// TIA Portal V17 export
// export: Created 2023-12-22T15:04:45.0691271Z, ExportSetting WithDefaults, DisplayName Totally Integrated Automation Portal, DisplayVersion V17, DisplayName TIA Portal Openness, DisplayVersion V17, DisplayName TIA Portal Version Control Interface, DisplayVersion V17, DisplayName STEP 7 Professional, DisplayVersion V17, DisplayName STEP 7 Safety, DisplayVersion V17, DisplayName WinCC Advanced, DisplayVersion V17
DATA_BLOCK "Main_Logick_DB"   // DB1
VERSION : 0.1
// stored: AutoNumber true, DBAccessibleFromOPCUA true, InstanceOfName Main_Logick, InstanceOfType FB
"Main_Logick"
   // VAR RETAIN
   //    Start : Bool;
   //    Start_Local : Bool;
   //    REQ_Pump : Bool;
   //    ev : Bool;
   //    Ready : Bool;
   //    Local : Bool;
   //    Mode : Bool;
   //    SP_Pump { S7_SetPoint := 'True'} : Real := 0.0;
   //    RM : Real;
   //    RM_SP { S7_SetPoint := 'True'} : Real := 0.0;
   //    Level_Norm { S7_SetPoint := 'True'} : Real := 50.0;
   //    Distance { S7_SetPoint := 'True'} : Real := 500.0;
   //    LE_Bar : Real;
   //    LE_Skvaz { S7_SetPoint := 'True'} : Real := 100.0;
   //    LE_Skvaz_RCHV { S7_SetPoint := 'True'} : Real := 0.0;
   //    Effect : Real;
   //    Alarm : Word;
   //    Alarms : Struct
   //       Leak : Bool;
   //       Level_Norm : Bool;
   //       LE_Warning : Bool;
   //       LE_Alarm : Bool;
   //    END_STRUCT;
   //    PID_Pump { S7_SetPoint := 'True'} : "PID_ex";
   // END_VAR
BEGIN
   PID_Pump.CMD.Vector := FALSE;
   PID_Pump.x := 1.0;
   PID_Pump.Settings.SP_P := 1.5;
   PID_Pump.Settings.SP_Ti := 150.0;
   PID_Pump.Settings.SP_Td := 0.0;
   PID_Pump.Settings.SP_Cycle := 0.2;
   PID_Pump.Settings.Max_SP := 500.0;
   PID_Pump.Settings.Min_SP := -500.0;
   PID_Pump.Settings.Max_in := 500.0;
   PID_Pump.Settings.Min_in := -500.0;
   PID_Pump.Settings.Max_out := 100.0;
   PID_Pump.Settings.Min_out := 0.0;
   PID_Pump.Settings.DeadBand := 1.0;
   PID_Pump.PID.IntegralResetMode := 4;
   PID_Pump.PID.RunModeByStartup := TRUE;
   PID_Pump.PID.SetSubstituteOutput := TRUE;
   PID_Pump.PID.ActivateRecoverMode := TRUE;
   PID_Pump.PID.CancelTuningLevel := 10.0;
   PID_Pump.PID.SubstituteOutput := 0.0;
   PID_Pump.PID.Config.InputPerOn := TRUE;
   PID_Pump.PID.Config.InvertControl := FALSE;
   PID_Pump.PID.Config.InputUpperLimit := 120.0;
   PID_Pump.PID.Config.InputLowerLimit := 0.0;
   PID_Pump.PID.Config.InputUpperWarning := 3.402822E+38;
   PID_Pump.PID.Config.InputLowerWarning := -3.402822E+38;
   PID_Pump.PID.Config.OutputUpperLimit := 100.0;
   PID_Pump.PID.Config.OutputLowerLimit := 0.0;
   PID_Pump.PID.Config.SetpointUpperLimit := 3.402822E+38;
   PID_Pump.PID.Config.SetpointLowerLimit := -3.402822E+38;
   PID_Pump.PID.Config.MinimumOnTime := 0.0;
   PID_Pump.PID.Config.MinimumOffTime := 0.0;
   PID_Pump.PID.Config.InputScaling.UpperPointIn := 27648.0;
   PID_Pump.PID.Config.InputScaling.LowerPointIn := 0.0;
   PID_Pump.PID.Config.InputScaling.UpperPointOut := 100.0;
   PID_Pump.PID.Config.InputScaling.LowerPointOut := 0.0;
   PID_Pump.PID.CycleTime.EnEstimation := TRUE;
   PID_Pump.PID.CycleTime.EnMonitoring := TRUE;
   PID_Pump.PID.CycleTime.Value := 0.1;
   PID_Pump.PID.CtrlParamsBackUp.Gain := 1.0;
   PID_Pump.PID.CtrlParamsBackUp.Ti := 20.0;
   PID_Pump.PID.CtrlParamsBackUp.Td := 0.0;
   PID_Pump.PID.CtrlParamsBackUp.TdFiltRatio := 0.2;
   PID_Pump.PID.CtrlParamsBackUp.PWeighting := 1.0;
   PID_Pump.PID.CtrlParamsBackUp.DWeighting := 1.0;
   PID_Pump.PID.CtrlParamsBackUp.Cycle := 1.0;
   PID_Pump.PID.PIDSelfTune.SUT.TuneRule := 0;
   PID_Pump.PID.PIDSelfTune.TIR.TuneRule := 0;
   PID_Pump.PID.Retain.CtrlParams.Gain := 1.0;
   PID_Pump.PID.Retain.CtrlParams.Ti := 20.0;
   PID_Pump.PID.Retain.CtrlParams.Td := 0.0;
   PID_Pump.PID.Retain.CtrlParams.TdFiltRatio := 0.2;
   PID_Pump.PID.Retain.CtrlParams.PWeighting := 1.0;
   PID_Pump.PID.Retain.CtrlParams.DWeighting := 1.0;
   PID_Pump.PID.Retain.CtrlParams.Cycle := 1.0;
   PID_Pump.C.SP := 1.0;
   PID_Pump.C.One := 0.1;
END_DATA_BLOCK
